(*
SPDX-FileCopyrightText: © 2026 Oleksandr Tiutyk <trofimich@gmail.com>
SPDX-License-Identifier: MIT
License: https://opensource.org/license/mit
*)

(*!
<summary>Exposes a borrowed view of the native open-file block owned by a resource manager.</summary>
<description>
This object owns neither the native block nor its handle. Keep the referenced FB_FileOpen alive for the entire
use of this view. The getters do not check acquisition: an assigned view is not evidence of an open file. Use
handle and target together only during the current acquisition, never after release. An invalid native-block
reference yields default scalar results or an invalid FilePath reference. Do not modify FilePath through its
reference, close the handle independently or delete this borrowed object.
</description>
*)

{attribute 'no_explicit_call' := 'Direct call is not allowed'}
FUNCTION_BLOCK INTERNAL FileHandleResource EXTENDS TOF_Core.Object
VAR_STAT
	//! <summary>Class name shared by all instances of this function block.</summary>
	{attribute 'hide'} 
	_ClassName : STRING := __POUNAME();
END_VAR
VAR
	{attribute 'hide'} 
	_FileOpen : REFERENCE TO Tc2_System.FB_FileOpen;
END_VAR

(*!
<summary>Target of the open file; use together with FileHandle.</summary>
*)

{attribute 'monitoring' := 'call'}

PROPERTY AmsNetId : Tc2_System.T_AmsNetID
GET
IF __ISVALIDREF(_FileOpen) THEN
	AmsNetId := _FileOpen.sNetId;
END_IF
END_GET
END_PROPERTY

(*!
<summary>Provides the concrete type name used in diagnostics.</summary>
<description>
Returns borrowed read-only metadata; keep the instance alive and do not modify the referenced string.
Reading does not allocate memory, initialize resources or transfer ownership.
</description>
*)
{attribute 'monitoring' := 'call'}
PROPERTY ClassName : REFERENCE TO STRING
GET
ClassName REF= _ClassName;
END_GET
END_PROPERTY

(*!
<summary>Binds this view to a caller-owned native file-open block without acquiring a file.</summary>
<description>
The binding is borrowed and must remain alive throughout use. An invalid reference is retained without
throwing; getters then return default scalars or an invalid reference. No handle is opened or closed.
</description>
<param name="fileOpen">Borrowed native block providing the path, target and current handle.</param>
*)
METHOD FB_Init: BOOL
VAR_INPUT
	bInitRetains : BOOL; // TRUE: the retain variables are initialized (reset warm / reset cold)
	bInCopyCode : BOOL;  // TRUE: the instance will be copied to the copy code afterward (online change)
	fileOpen : REFERENCE TO Tc2_System.FB_FileOpen;
END_VAR
_FileOpen REF= fileOpen;
END_METHOD

(*!
<summary>Reads the native handle from the borrowed open-file block.</summary>
<description>
Returns the default UINT when no native block is bound. Does not check acquisition or close status; a stored
numeric handle must not be reused after release.
</description>
*)
{attribute 'monitoring' := 'call'}
PROPERTY FileHandle : UINT
GET
IF __ISVALIDREF(_FileOpen) THEN
	FileHandle := _FileOpen.hFile;
END_IF
END_GET
END_PROPERTY

(*!
<summary>Provides a borrowed view of the configured native file path.</summary>
<description>
The reference is invalid when no native block is bound. Keep the owner alive and do not write through this
reference. This path identifies configuration, not proof that the file is open.
</description>
*)
{attribute 'monitoring' := 'call'}
PROPERTY FilePath : REFERENCE TO Tc2_System.T_MaxString
GET
IF __ISVALIDREF(_FileOpen) THEN
	FilePath REF= _FileOpen.sPathName;
END_IF
END_GET
END_PROPERTY

(*!
<summary>Provides the library namespace used in diagnostics.</summary>
<description>Returns borrowed read-only namespace storage; do not modify the referenced string.</description>
*)
{attribute 'monitoring' := 'call'}
PROPERTY NamespaceName : REFERENCE TO STRING
GET
NamespaceName REF= CurrentNamespace.Name;
END_GET
END_PROPERTY

(*!
<summary>Reports the size of this concrete instance in bytes.</summary>
*)
{attribute 'monitoring' := 'call'}
PROPERTY SelfSize : ULINT
GET
SelfSize := XSIZEOF(THIS^);
END_GET
END_PROPERTY

END_FUNCTION_BLOCK

(* stored: Version 1.1.0.1
   POU FileHandleResource: Id {3b5c26cf-3170-4545-bd8c-3bd2c4df1329}, SpecialFunc None
   Property AmsNetId: Id {380802f5-49e1-48ab-848f-8d4221f7487f}
   Get Get: Id {6426ac28-9518-4d34-82d5-0cb3445bd540}
   Property ClassName: Id {e357a305-e7de-4b32-92a8-00371949d47e}
   Get Get: Id {284aba92-edd1-4b1b-9361-0330fa8f6d0c}
   Method FB_Init: Id {3a7a9b22-aecf-4b7b-98d9-39fda05e6a70}
   Property FileHandle: Id {41387944-3b27-40d9-a71a-79172bcfc3c1}
   Get Get: Id {5c0a725f-80b2-4645-9072-3dcfb1a89456}
   Property FilePath: Id {b9868a13-98bb-41c4-aa60-43cac9371bda}
   Get Get: Id {97ff0fdc-ec21-47e3-8ff8-51dd09c647a3}
   Property NamespaceName: Id {4f8fd457-4527-453a-bb0a-b797e3616ec8}
   Get Get: Id {a13f030a-2ce4-4068-b49d-03db3751d4f0}
   Property SelfSize: Id {18c8a656-741c-413f-993f-ac37337ec5cd}
   Get Get: Id {79dc3c1f-cd1f-4f38-b451-48654d0e5843} *)
